(* CODESYS project Storage2018v1.project

Project tree, tasks and I/O mapping:
  CODESYS_Control_Win_V3_x64 : CODESYS Control Win V3 x64, 3S - Smart Software Solutions GmbH, version 3.5.12.30
    application Application
      libraries: BASIC, 3.31 (OSCAT)
      task VISU_TASK (cyclic, interval 50 ms, priority 31) calls VisuElems.Visu_Prg
      task Task (cyclic, interval t#20ms, priority 1) calls main, simulationLogic
      Control/
        program main [ST]
        Support/
          data type Position
          data type ArmRequest
          data type OPState
          function block ButtonRequester [LD]
          function PosToButtons [ST]
          function ButtonsToPos [ST]
          function block ArmRequestHandler [LD]
        program ArmControl [LD]
        function block PositionState [LD]
        function block OPArmMover [LD]
        function block OPGripper [SFC]
        function block OPPickNPlace [SFC]: copyVariables, gotoPos
        function block OPpnpTester [SFC]: setPick1, setPick2, setPick3, setPlace1, setPlace2, setPlace3
      doNotChange/
        Components/
          program simulationLogic [ST]
          visualisation armNStore
          Storage/
            visualisation StoragePlace
            visualisation Storage
            program storageLogic [ST]
          Conveyor/
            visualisation Conveyor
            program conveyorLogic [ST]
          Arm/
            visualisation TheArm
            program armLogic [ST]
            visualisation Gripper
        SimulationHelpers/
          function block MoveObject [ST]
        global variables InternalSimulation
        IO and DataTypes/
          data type CylPos
          data type XYPos
          data type ArmCommand
        internalTypes/
          data type StoragePos
        program simulationMapping [ST]
      Simulation/
        visualisation Simulation
      global variables IOs
  libraries: SysTimeCore, 3.5.5.0 (System)
  text list GlobalTextList
*)

// CODESYS_Control_Win_V3_x64/Application/Control/Support/Position
TYPE Position :
STRUCT
	x: INT;
	y: INT;
END_STRUCT
END_TYPE

// CODESYS_Control_Win_V3_x64/Application/Control/Support/ArmRequest
TYPE ArmRequest :
STRUCT
	run: BOOL;
	goto: Position;
END_STRUCT
END_TYPE

// CODESYS_Control_Win_V3_x64/Application/Control/Support/OPState
TYPE OPState :
STRUCT
	initial: BOOL;
	executing: BOOL;
	finished: BOOL;
END_STRUCT
END_TYPE

// CODESYS_Control_Win_V3_x64/Application/doNotChange/IO and DataTypes/CylPos
TYPE CylPos :
	STRUCT
		occupied: BOOL;
		id: STRING;
	END_STRUCT
END_TYPE

// CODESYS_Control_Win_V3_x64/Application/doNotChange/IO and DataTypes/XYPos
TYPE XYPos :
	STRUCT
		posX: INT;
		posY: INT;
	END_STRUCT
END_TYPE

// CODESYS_Control_Win_V3_x64/Application/doNotChange/IO and DataTypes/ArmCommand
TYPE ArmCommand :
STRUCT
	fromPos: XYPos;
	toPos: XYPos;
END_STRUCT
END_TYPE

// CODESYS_Control_Win_V3_x64/Application/doNotChange/internalTypes/StoragePos
TYPE StoragePos :
	STRUCT
		cyl: CylPos;
		pos: XYPos;
		pressed: Bool;
	END_STRUCT
END_TYPE

// CODESYS_Control_Win_V3_x64/Application/doNotChange/InternalSimulation
VAR_GLOBAL
	error: BOOL := FALSE;
	errorText: STRING := '';
	disablePressPos: BOOL := FALSE;
	buttonUP: BOOL;
	buttonDown: BOOL;
	buttonRun: BOOL;
	buttonDir: BOOL;
	buttonExt: BOOL;
	buttonRetr: BOOL;
	buttonGrip: BOOL;
END_VAR

// CODESYS_Control_Win_V3_x64/Application/IOs
VAR_GLOBAL
	qxArmRun: BOOL := FALSE; // Starts the arm moving left and right
	qxArmDirection: BOOL := FALSE; // true -> left, false -> right
	qxArmUp: BOOL := FALSE; // moves the arm up
	qxArmDown: BOOL := FALSE; // moves the arm down
	qxGripExtend: BOOL := FALSE; // extends the gripper
	qxGripRetract: BOOL := FALSE; // retracts the gripper
	qxGripping: BOOL := FALSE; // releases when false
	qxPosLamp: ARRAY[0..2, 0..2] OF BOOL;// lamp[X, Y] control if on / off
	
	ixArmAtX0: BOOL := FALSE;	// The arm postion
	ixArmAtX1: BOOL := FALSE;
	ixArmAtX2: BOOL := FALSE;
	ixArmAtY0: BOOL := FALSE;
	ixArmAtY1: BOOL := FALSE;
	ixArmAtY2: BOOL := FALSE;
	ixPosButtonDown: ARRAY[0..2, 0..2] OF BOOL;// Button[X, Y] is currently beeing pressed
	
	// These may not be the same as the qx versions above since the 
	// buttons in the simulation also can control the motion
	ixArmRun: BOOL := FALSE; // If the arm is moving left or rigth
	ixArmDirection: BOOL := FALSE; // true -> left, false -> right
	ixArmUp: BOOL := FALSE; // if arm is moving up
	ixArmDown: BOOL := FALSE; // if the arm is moving down
	
	ixGripExtended: BOOL := FALSE;	// the gripper has been extended
	ixGripRetracted: BOOL := FALSE; // the gripper has been retracted
	ixCylinderInGripper: BOOL:=FALSE; // A cylinder is carried by the arm
	
	ixEmergency: BOOL := TRUE; // Emergency stop if value is false
	ixStartButton: BOOL := FALSE;
	ixRunSequence: bool:= false;
		
END_VAR

// CODESYS_Control_Win_V3_x64/Application/Control/main
PROGRAM main
VAR

END_VAR

ArmControl();

END_PROGRAM

// CODESYS_Control_Win_V3_x64/Application/Control/ArmControl
PROGRAM ArmControl
VAR

	goto1: BOOL;
	goto0: BOOL;
	goto2: BOOL;
	
	initial: BOOL := FALSE;
	PositionStateY: PositionState;
	armYPosition: INT;
	armXPosition: INT;
	PositionStateX: PositionState;
	buttonReq: ButtonRequester;
	armMover: OPArmMover;
	moveRight: BOOL;
	moveLeft: BOOL;
	armGripper: OPGripper;
	reqHandler: ArmRequestHandler;
	pickNPlace: OPPickNPlace;
	staticPos: Position := (x := 3, y := 3);
	pnpTester: OPpnpTester;
END_VAR

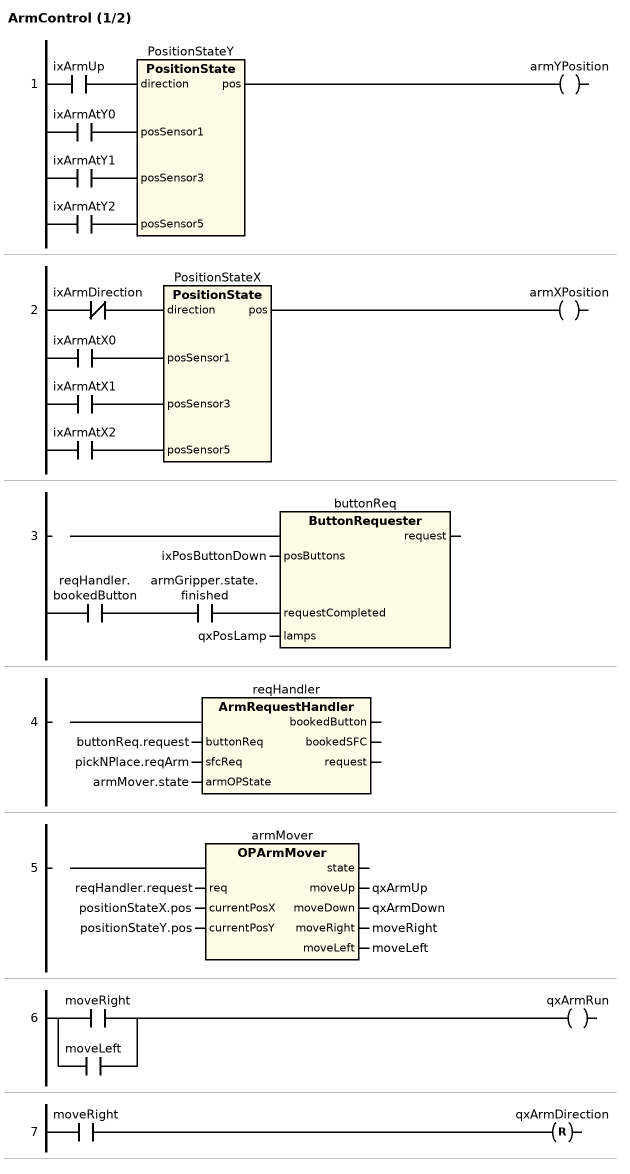
// NETWORK 1
PositionStateY(
    direction := ixArmUp,
    posSensor1 := ixArmAtY0,
    posSensor3 := ixArmAtY1,
    posSensor5 := ixArmAtY2); // PositionState
armYPosition := PositionStateY.pos;

// NETWORK 2
PositionStateX(
    direction := NOT ixArmDirection,
    posSensor1 := ixArmAtX0,
    posSensor3 := ixArmAtX1,
    posSensor5 := ixArmAtX2); // PositionState
armXPosition := PositionStateX.pos;

// NETWORK 3
buttonReq(
    posButtons := ixPosButtonDown,
    requestCompleted := reqHandler.bookedButton AND armGripper.state.finished,
    lamps := qxPosLamp); // ButtonRequester

// NETWORK 4
reqHandler(buttonReq := buttonReq.request, sfcReq := pickNPlace.reqArm, armOPState := armMover.state); // ArmRequestHandler

// NETWORK 5
armMover(
    req := reqHandler.request,
    currentPosX := positionStateX.pos,
    currentPosY := positionStateY.pos,
    moveUp => qxArmUp,
    moveDown => qxArmDown,
    moveRight => moveRight,
    moveLeft => moveLeft); // OPArmMover

// NETWORK 6
qxArmRun := moveRight OR moveLeft;

// NETWORK 7
qxArmDirection R= moveRight;

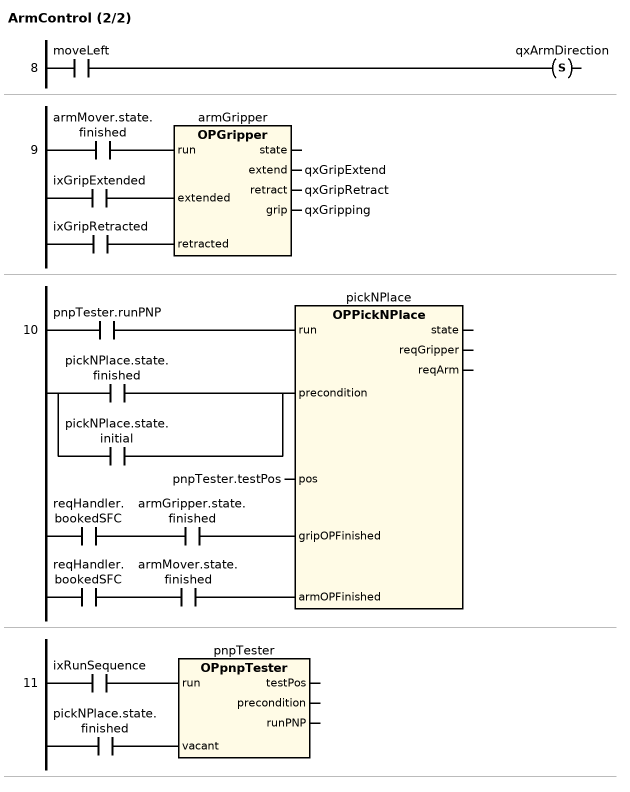
// NETWORK 8
qxArmDirection S= moveLeft;

// NETWORK 9
armGripper(
    run := armMover.state.finished,
    extended := ixGripExtended,
    retracted := ixGripRetracted,
    extend => qxGripExtend,
    retract => qxGripRetract,
    grip => qxGripping); // OPGripper

// NETWORK 10
pickNPlace(
    run := pnpTester.runPNP,
    precondition := pickNPlace.state.finished OR pickNPlace.state.initial,
    pos := pnpTester.testPos,
    gripOPFinished := reqHandler.bookedSFC AND armGripper.state.finished,
    armOPFinished := reqHandler.bookedSFC AND armMover.state.finished); // OPPickNPlace

// NETWORK 11
pnpTester(run := ixRunSequence, vacant := pickNPlace.state.finished); // OPpnpTester

END_PROGRAM

// CODESYS_Control_Win_V3_x64/Application/Control/PositionState
FUNCTION_BLOCK PositionState
VAR_INPUT
	direction: BOOL;
	posSensor1: BOOL;
	posSensor3: BOOL;
	posSensor5: BOOL;
END_VAR
VAR_OUTPUT
	pos: INT := -1;
END_VAR
VAR
	trig: F_TRIG;
END_VAR

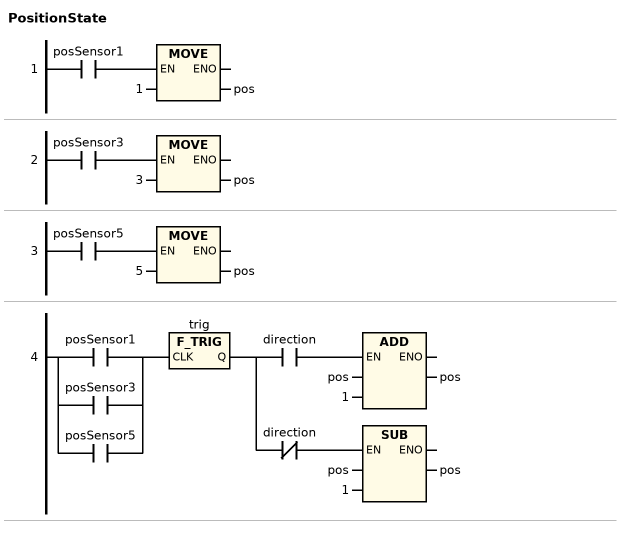
// NETWORK 1
IF posSensor1 THEN pos := 1; END_IF

// NETWORK 2
IF posSensor3 THEN pos := 3; END_IF

// NETWORK 3
IF posSensor5 THEN pos := 5; END_IF

// NETWORK 4
trig(CLK := posSensor1 OR posSensor3 OR posSensor5); // F_TRIG
IF trig.Q AND direction THEN pos := pos + 1; END_IF
IF trig.Q AND NOT direction THEN pos := pos - 1; END_IF

END_FUNCTION_BLOCK

// CODESYS_Control_Win_V3_x64/Application/Control/Support/ButtonRequester
FUNCTION_BLOCK ButtonRequester
VAR_INPUT
	posButtons: ARRAY[0..2, 0..2] OF BOOL;
	requestCompleted: BOOL;
END_VAR
VAR_OUTPUT
	request: ArmRequest;
END_VAR
VAR_IN_OUT
	lamps: ARRAY[0..2, 0..2] OF BOOL;
END_VAR

VAR
	armPos: Position;
	buttX: INT;
	buttY: INT;
	buttonPressed: BOOL;
	noRequest: ArmRequest := (run:=FALSE, goto := (x:=-1, y:=-1));
END_VAR
VAR // added by the converter: edge detectors and wires of the graphical bodies
    _w1 : BOOL;
END_VAR

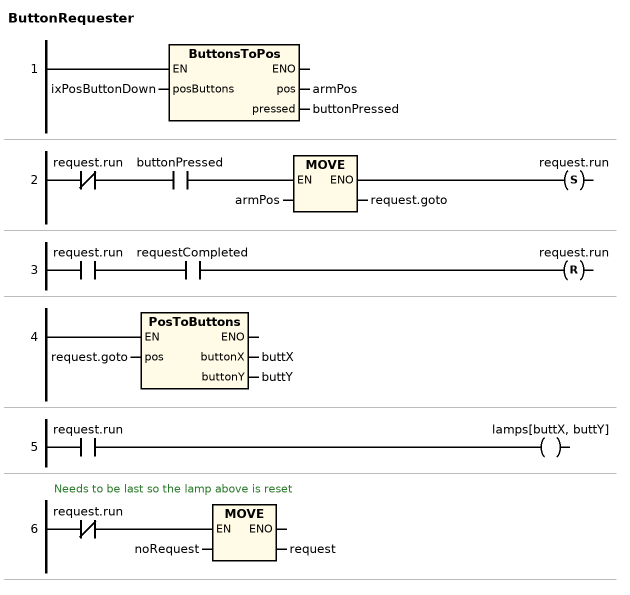
// NETWORK 1
ButtonsToPos(posButtons := ixPosButtonDown, pos => armPos, pressed => buttonPressed);

// NETWORK 2
_w1 := NOT request.run AND buttonPressed;
IF _w1 THEN request.goto := armPos; END_IF
request.run S= _w1;

// NETWORK 3
request.run R= request.run AND requestCompleted;

// NETWORK 4
PosToButtons(pos := request.goto, buttonX => buttX, buttonY => buttY);

// NETWORK 5
lamps[buttX, buttY] := request.run;

// NETWORK 6
// Needs to be last so the lamp above is reset
IF NOT request.run THEN request := noRequest; END_IF

END_FUNCTION_BLOCK

// CODESYS_Control_Win_V3_x64/Application/Control/Support/ButtonsToPos
FUNCTION ButtonsToPos
VAR_INPUT
	posButtons: ARRAY[0..2, 0..2] OF BOOL;
END_VAR
VAR_OUTPUT
	pos: Position;
	pressed: BOOL;
END_VAR
VAR
	x: INT;
	y: INT;
END_VAR

pos.x := -1;
pos.y := -1;
pressed := FALSE;

FOR x:=0 TO 2 DO
	FOR y:=0 TO 2 DO
		IF posButtons[x,y] THEN
			pos.x := 1 + x*2;
			pos.y := 1 + y*2;
			pressed := TRUE;
		END_IF
	END_FOR
END_FOR

END_FUNCTION

// CODESYS_Control_Win_V3_x64/Application/Control/Support/PosToButtons
FUNCTION PosToButtons
VAR_INPUT
	pos: Position;
END_VAR
VAR_OUTPUT
	buttonX: INT;
	buttonY: INT;
END_VAR
VAR
END_VAR

buttonX := -1;
buttonY := -1;
IF EVEN(pos.x-1) AND EVEN(pos.y-1) THEN
	buttonX:= (pos.x-1)/2;
	buttonY:= (pos.y-1)/2;
END_IF

END_FUNCTION

// CODESYS_Control_Win_V3_x64/Application/Control/Support/ArmRequestHandler
FUNCTION_BLOCK ArmRequestHandler
VAR_INPUT
	buttonReq: ArmRequest;
	sfcReq: ArmRequest;
	armOPState: OPState;
END_VAR
VAR_OUTPUT
	bookedButton: BOOL;
	bookedSFC: BOOL;
	request: ArmRequest;
END_VAR
VAR
	noRequest: ArmRequest := (run:=FALSE, goto := (x:=-1, y:=-1));
END_VAR

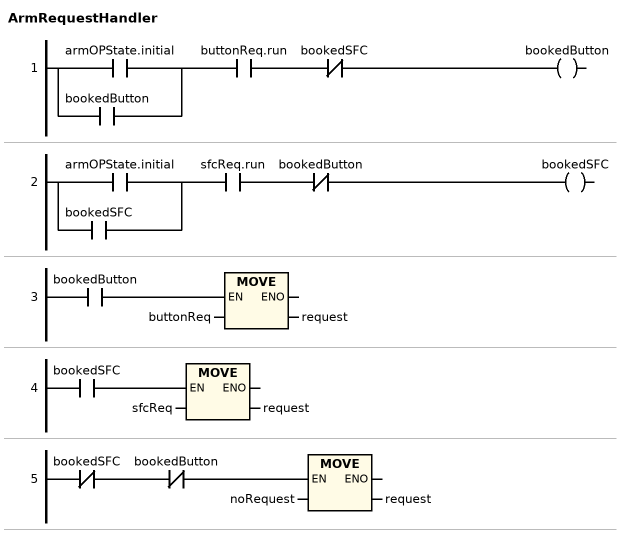
// NETWORK 1
bookedButton := (armOPState.initial OR bookedButton) AND buttonReq.run AND NOT bookedSFC;

// NETWORK 2
bookedSFC := (armOPState.initial OR bookedSFC) AND sfcReq.run AND NOT bookedButton;

// NETWORK 3
IF bookedButton THEN request := buttonReq; END_IF

// NETWORK 4
IF bookedSFC THEN request := sfcReq; END_IF

// NETWORK 5
IF NOT bookedSFC AND NOT bookedButton THEN request := noRequest; END_IF

END_FUNCTION_BLOCK

// CODESYS_Control_Win_V3_x64/Application/Control/OPArmMover
FUNCTION_BLOCK OPArmMover
VAR_INPUT
	req: ArmRequest;
	currentPosX: INT;
	currentPosY: INT;
END_VAR
VAR_OUTPUT
	state: OPState := (	initial := TRUE, 
						executing := FALSE, 
						finished := FALSE);
	moveUp: BOOL;
	moveDown: BOOL;
	moveRight: BOOL;
	moveLeft: BOOL;
END_VAR
VAR
	
	gotoX: INT;
	gotoY: INT;
	R_TRIG_0: R_TRIG;
	F_TRIG_0: F_TRIG;
	armGripper: OPGripper;
END_VAR
VAR // added by the converter: edge detectors and wires of the graphical bodies
    _w1, _w2 : BOOL;
END_VAR

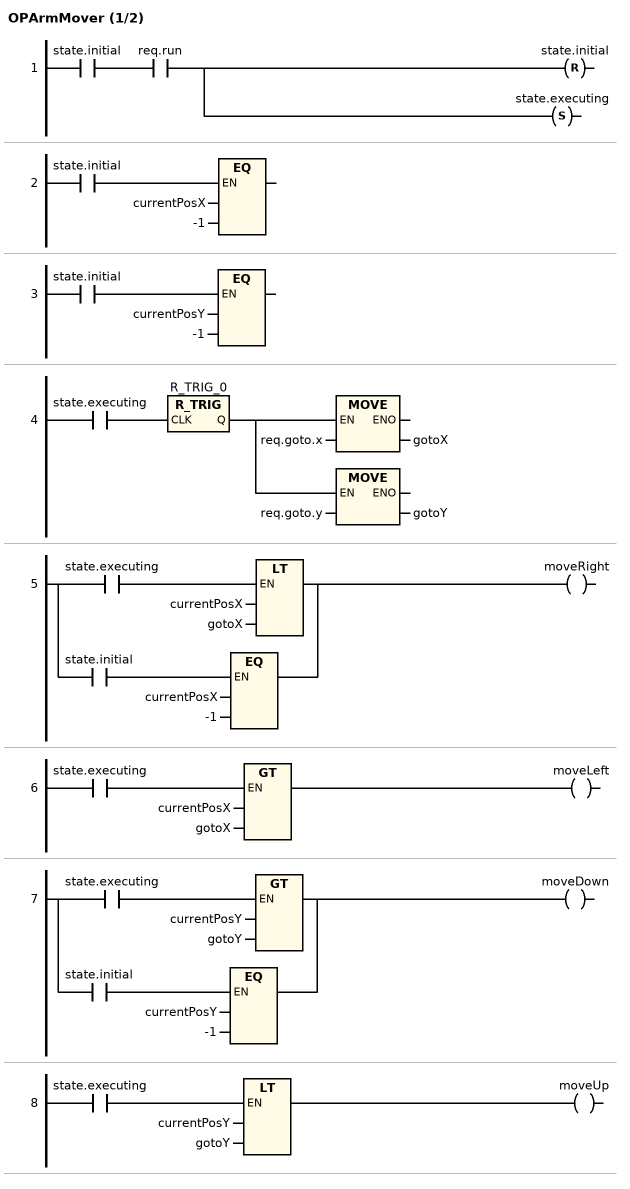
// NETWORK 1
_w1 := state.initial AND req.run;
state.initial R= _w1;
state.executing S= _w1;

// NETWORK 2
(* state.initial AND currentPosX = -1; result not used *)

// NETWORK 3
(* state.initial AND currentPosY = -1; result not used *)

// NETWORK 4
R_TRIG_0(CLK := state.executing); // R_TRIG
IF R_TRIG_0.Q THEN gotoX := req.goto.x; END_IF
IF R_TRIG_0.Q THEN gotoY := req.goto.y; END_IF

// NETWORK 5
moveRight := state.executing AND currentPosX < gotoX OR state.initial AND currentPosX = -1;

// NETWORK 6
moveLeft := state.executing AND currentPosX > gotoX;

// NETWORK 7
moveDown := state.executing AND currentPosY > gotoY OR state.initial AND currentPosY = -1;

// NETWORK 8
moveUp := state.executing AND currentPosY < gotoY;

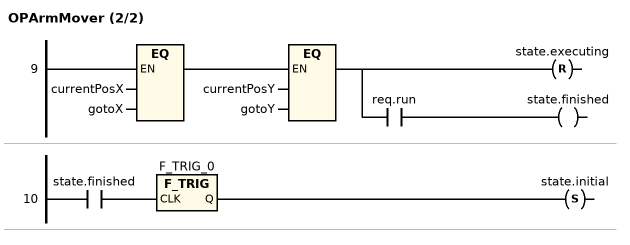
// NETWORK 9
_w2 := currentPosX = gotoX AND currentPosY = gotoY;
state.executing R= _w2;
state.finished := _w2 AND req.run;

// NETWORK 10
F_TRIG_0(CLK := state.finished); // F_TRIG
state.initial S= F_TRIG_0.Q;

END_FUNCTION_BLOCK

// CODESYS_Control_Win_V3_x64/Application/Control/OPGripper
FUNCTION_BLOCK OPGripper
VAR_INPUT
	run: BOOL;
	extended: BOOL;
	retracted: BOOL;
END_VAR
VAR_OUTPUT
	state: OPState;
	extend: BOOL;
	retract: BOOL;
	grip: BOOL;
END_VAR
VAR
END_VAR

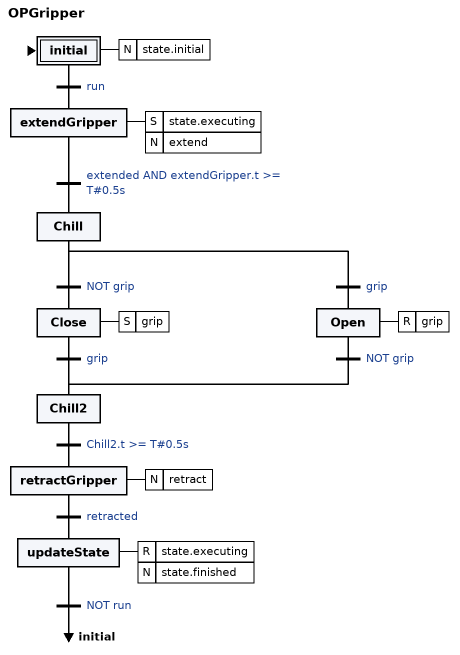
INITIAL_STEP initial:
    state.initial(N);
END_STEP
TRANSITION FROM initial TO extendGripper
    := run;
END_TRANSITION
STEP extendGripper:
    state.executing(S);
    extend(N);
END_STEP
TRANSITION FROM extendGripper TO Chill
    := extended AND extendGripper.t >= T#0.5s;
END_TRANSITION
STEP Chill:
END_STEP
TRANSITION FROM Chill TO Close
    := NOT grip;
END_TRANSITION
STEP Close:
    grip(S);
END_STEP
TRANSITION FROM Close TO Chill2
    := grip;
END_TRANSITION
TRANSITION FROM Chill TO Open
    := grip;
END_TRANSITION
STEP Open:
    grip(R);
END_STEP
TRANSITION FROM Open TO Chill2
    := NOT grip;
END_TRANSITION
STEP Chill2:
END_STEP
TRANSITION FROM Chill2 TO retractGripper
    := Chill2.t >= T#0.5s;
END_TRANSITION
STEP retractGripper:
    retract(N);
END_STEP
TRANSITION FROM retractGripper TO updateState
    := retracted;
END_TRANSITION
STEP updateState:
    state.executing(R);
    state.finished(N);
END_STEP
TRANSITION FROM updateState TO initial
    := NOT run;
END_TRANSITION

END_FUNCTION_BLOCK

// CODESYS_Control_Win_V3_x64/Application/Control/OPPickNPlace
FUNCTION_BLOCK OPPickNPlace
VAR_INPUT
	run: BOOL;
	precondition: BOOL;
	pos: Position;
	gripOPFinished: BOOL;
	armOPFinished: BOOL;
END_VAR
VAR_OUTPUT
	state: OPState;
	reqGripper: BOOL;
	reqArm: ArmRequest;
END_VAR
VAR
END_VAR

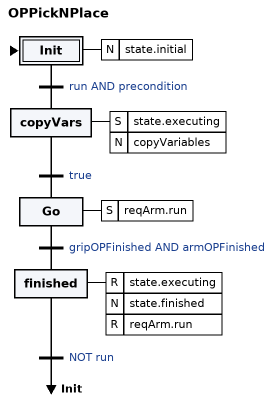
INITIAL_STEP Init:
    state.initial(N);
END_STEP
TRANSITION FROM Init TO copyVars
    := run AND precondition;
END_TRANSITION
STEP copyVars:
    state.executing(S);
    copyVariables(N);
END_STEP
TRANSITION FROM copyVars TO Go
    := true;
END_TRANSITION
STEP Go:
    reqArm.run(S);
END_STEP
TRANSITION FROM Go TO finished
    := gripOPFinished AND armOPFinished;
END_TRANSITION
STEP finished:
    state.executing(R);
    state.finished(N);
    reqArm.run(R);
END_STEP
TRANSITION FROM finished TO Init
    := NOT run;
END_TRANSITION

ACTION copyVariables:

(* Copy destination position *)
reqArm.goto.x := pos.x;
reqArm.goto.y := pos.y;
END_ACTION

ACTION gotoPos:
reqArm.run := true;
END_ACTION

END_FUNCTION_BLOCK

// CODESYS_Control_Win_V3_x64/Application/Control/OPpnpTester
FUNCTION_BLOCK OPpnpTester
VAR_INPUT
	run: BOOL;
	vacant: BOOL;
END_VAR
VAR_OUTPUT
	testPos: Position;
	precondition: BOOL;
	runPNP: BOOL;
END_VAR
VAR
	pick1: Position := (x := 1, y := 3);
	place1: Position := (x := 5, y := 5);
	
	pick2: Position := (x := 5, y := 1);
	place2: Position := (x := 3, y := 3);
	
	pick3: Position := (x := 3, y := 3);
	place3: Position := (x := 1, y := 5);
END_VAR

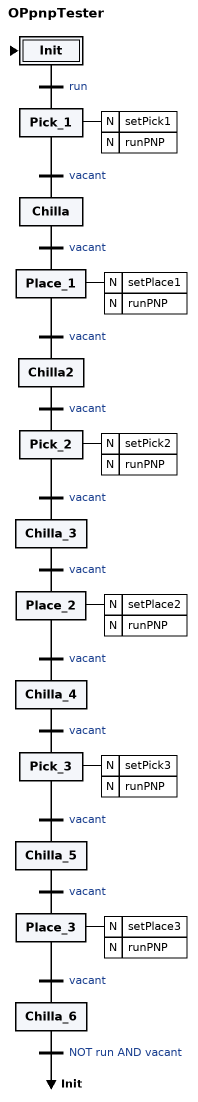
INITIAL_STEP Init:
END_STEP
TRANSITION FROM Init TO Pick_1
    := run;
END_TRANSITION
STEP Pick_1:
    setPick1(N);
    runPNP(N);
END_STEP
TRANSITION FROM Pick_1 TO Chilla
    := vacant;
END_TRANSITION
STEP Chilla:
END_STEP
TRANSITION FROM Chilla TO Place_1
    := vacant;
END_TRANSITION
STEP Place_1:
    setPlace1(N);
    runPNP(N);
END_STEP
TRANSITION FROM Place_1 TO Chilla2
    := vacant;
END_TRANSITION
STEP Chilla2:
END_STEP
TRANSITION FROM Chilla2 TO Pick_2
    := vacant;
END_TRANSITION
STEP Pick_2:
    setPick2(N);
    runPNP(N);
END_STEP
TRANSITION FROM Pick_2 TO Chilla_3
    := vacant;
END_TRANSITION
STEP Chilla_3:
END_STEP
TRANSITION FROM Chilla_3 TO Place_2
    := vacant;
END_TRANSITION
STEP Place_2:
    setPlace2(N);
    runPNP(N);
END_STEP
TRANSITION FROM Place_2 TO Chilla_4
    := vacant;
END_TRANSITION
STEP Chilla_4:
END_STEP
TRANSITION FROM Chilla_4 TO Pick_3
    := vacant;
END_TRANSITION
STEP Pick_3:
    setPick3(N);
    runPNP(N);
END_STEP
TRANSITION FROM Pick_3 TO Chilla_5
    := vacant;
END_TRANSITION
STEP Chilla_5:
END_STEP
TRANSITION FROM Chilla_5 TO Place_3
    := vacant;
END_TRANSITION
STEP Place_3:
    setPlace3(N);
    runPNP(N);
END_STEP
TRANSITION FROM Place_3 TO Chilla_6
    := vacant;
END_TRANSITION
STEP Chilla_6:
END_STEP
TRANSITION FROM Chilla_6 TO Init
    := NOT run AND vacant;
END_TRANSITION

ACTION setPick1:


testPos.x := pick1.x;
testPos.y := pick1.y;
END_ACTION

ACTION setPick2:


testPos.x := pick2.x;
testPos.y := pick2.y;
END_ACTION

ACTION setPick3:


testPos.x := pick3.x;
testPos.y := pick3.y;
END_ACTION

ACTION setPlace1:


testPos.x := place1.x;
testPos.y := place1.y;
END_ACTION

ACTION setPlace2:


testPos.x := place2.x;
testPos.y := place2.y;
END_ACTION

ACTION setPlace3:


testPos.x := place3.x;
testPos.y := place3.y;
END_ACTION

END_FUNCTION_BLOCK

// CODESYS_Control_Win_V3_x64/Application/doNotChange/Components/simulationLogic
PROGRAM simulationLogic
VAR
	armAtX0: BOOL := FALSE;
	armAtX1: BOOL := FALSE;
	armAtX2: BOOL := FALSE;
	armAtY0: BOOL := FALSE;
	armAtY1: BOOL := FALSE;
	armAtY2: BOOL := FALSE;
	inAnyPos: BOOL := FALSE;
	graspTrig: R_TRIG;
	relTrig: F_TRIG;
	grasp: BOOL;
	release: BOOL;
	errorMsg: STRING := '';
	ack: BOOL:= FALSE;
	e_stop: BOOL:= FALSE;
	allowPick: BOOL;
END_VAR

storageLogic();
armLogic();
simulationMapping();

armAtX0 := armLogic.armPosX > 90 AND armLogic.armPosX < 95;
armAtX1 := armLogic.armPosX > 205 AND armLogic.armPosX < 210;
armAtX2 := armLogic.armPosX > 320 AND armLogic.armPosX < 325;

armAtY2 := armLogic.armPosY > 0 AND armLogic.armPosY < 15;
armAtY1 := armLogic.armPosY > 100 AND armLogic.armPosY < 115;
armAtY0 := armLogic.armPosY > 200 AND armLogic.armPosY < 215;

inAnyPos := (armAtX0 OR armAtX1 OR armAtX2) AND (armAtY0 OR armAtY1 OR armAtY2);
allowPick := inAnyPos AND ixGripExtended;

graspTrig(CLK:= qxGripping, Q=> grasp);
relTrig(CLK:= qxGripping, Q=> release);

IF grasp AND allowPick THEN
	ixCylinderInGripper := TRUE;
END_IF
IF release AND allowPick THEN
	ixCylinderInGripper := FALSE;
END_IF

// Error handling
IF e_stop AND ixEmergency THEN
	ixEmergency := FALSE;
	errorMsg := 'You pressed the Emergency';
END_IF
IF ack THEN
	ixEmergency := TRUE;
	errorMsg := '';
END_IF

IF grasp AND inAnyPos AND NOT allowPick AND ixEmergency THEN
	ixEmergency := FALSE;
	errorMsg := 'Not grasping when gripper is extended!';
ELSIF grasp AND NOT inAnyPos AND ixEmergency THEN
	ixEmergency := FALSE;
	errorMsg := 'Not grasping at a XY position!';
END_IF

IF release AND (NOT inAnyPos OR NOT ixGripExtended) AND ixEmergency AND ixCylinderInGripper THEN
	ixEmergency := FALSE;
	errorMsg := 'You dropped the cylinder';
	ixCylinderInGripper := FALSE;
END_IF

IF (qxArmRun OR qxArmDown OR qxArmUp) AND ixGripExtended THEN
	ixEmergency := FALSE;
	errorMsg := 'Can not move white extended gripper';
END_IF

END_PROGRAM

// CODESYS_Control_Win_V3_x64/Application/doNotChange/Components/Storage/storageLogic
PROGRAM storageLogic
VAR
	storagePlaces: ARRAY[0..2, 0..2] OF StoragePos;
END_VAR

	storageLogic.storagePlaces[0,0].cyl.occupied := qxPosLamp[0,0];
	storageLogic.storagePlaces[0,1].cyl.occupied := qxPosLamp[0,1];
	storageLogic.storagePlaces[0,2].cyl.occupied := qxPosLamp[0,2];
	storageLogic.storagePlaces[1,0].cyl.occupied := qxPosLamp[1,0];
	storageLogic.storagePlaces[1,1].cyl.occupied := qxPosLamp[1,1];
	storageLogic.storagePlaces[1,2].cyl.occupied := qxPosLamp[1,2];
	storageLogic.storagePlaces[2,0].cyl.occupied := qxPosLamp[2,0];
	storageLogic.storagePlaces[2,1].cyl.occupied := qxPosLamp[2,1];
	storageLogic.storagePlaces[2,2].cyl.occupied := qxPosLamp[2,2];

END_PROGRAM

// CODESYS_Control_Win_V3_x64/Application/doNotChange/Components/Arm/armLogic
PROGRAM armLogic
VAR
	gripping: BOOL := FALSE;
	extending: BOOL := FALSE;
	cyl: CylPos := (occupied := FALSE, id:= '');
	armPosX : INT;
	armPosY : INT;
	gripYPos: INT := 0;
	gripXPos: INT := 0;
	moveArm: MoveObject;
	armDown: BOOL := FALSE;
	armUP: BOOL := false;
	armL: BOOL := false;
	armR: BOOL := false;
END_VAR
VAR_TEMP
	
END_VAR

IF extending THEN
	gripYPos := -25;
ELSE
	gripYPos := 0;
END_IF
gripXPos := 0;

armLogic.cyl.occupied := ixCylinderInGripper;
IF ixCylinderInGripper THEN
	armLogic.cyl.id := 'Cylinder';
ELSE
	armLogic.cyl.id := '';
END_IF

moveArm(
	moveUP:= armUP, 
	moveDown:= armDown, 
	moveLeft:=armL , 
	moveRight:=armR , 
	maxX:=400, 
	minX:=0, 
	maxY:=220, 
	minY:=0, 
	tick:=T#0.01S , 
	x:= armPosX, 
	y:=armPosY );
	
	armLogic.armR := (qxArmRun AND NOT qxArmDirection) OR (buttonRun AND NOT buttonDir) ;
	armLogic.armL := (qxArmRun AND qxArmDirection) OR (buttonRun AND buttonDir);	
	armLogic.armUP := qxArmUp OR buttonUP;
	armLogic.armDown := qxArmDown OR buttonDown;
	armLogic.extending := qxGripExtend OR buttonExt OR (armLogic.extending AND NOT (qxGripRetract OR buttonRetr));
	armLogic.gripping := qxGripping OR buttonGrip;
	
	ixArmUp := armLogic.armUP;
	ixArmDown := armLogic.armDown;
	ixArmRun := qxArmRun OR buttonRun;
	ixArmDirection := qxArmDirection OR buttonDir;

END_PROGRAM

// CODESYS_Control_Win_V3_x64/Application/doNotChange/SimulationHelpers/MoveObject
FUNCTION_BLOCK MoveObject
VAR_INPUT
	moveUP: BOOL;
	moveDown: BOOL;
	moveLeft: BOOL;
	moveRight: BOOL;
	maxX: INT;
	minX: INT;
	maxY: INT;
	minY: INT;
	tick: time;
END_VAR
VAR_IN_OUT
	x: INT;
	y: INT;
END_VAR
VAR_OUTPUT
END_VAR
VAR
	pulse: clk_pulse;
END_VAR

pulse(
	PT:= tick, 
	N:= 0, 
	RST:= NOT moveUp AND NOT moveDown AND NOT moveLeft AND NOT moveRight , 
	Q=> , 
	CNT=> , 
	RUN=> );
	
IF pulse.Q THEN
	IF moveUP AND NOT moveDown AND y > minY THEN
		y := y-1;
	ELSIF NOT moveUP AND moveDown AND y < maxY THEN
		y := y+1;
	END_IF
	
	IF moveRight AND NOT moveLeft AND x < maxX THEN
		x := x+1;
	ELSIF NOT moveRight AND moveLeft AND x > minX THEN
		x := x-1;
	END_IF
END_IF

END_FUNCTION_BLOCK

// CODESYS_Control_Win_V3_x64/Application/doNotChange/simulationMapping
PROGRAM simulationMapping
VAR
END_VAR



	

	
	
	ixArmAtX0 := simulationLogic.armAtX0;
	ixArmAtX1 := simulationLogic.armAtX1;
	ixArmAtX2 := simulationLogic.armAtX2;
	ixArmAtY0 := simulationLogic.armAtY0;
	ixArmAtY1 := simulationLogic.armAtY1;
	ixArmAtY2 := simulationLogic.armAtY2;
	ixPosButtonDown[0,0] := storageLogic.storagePlaces[0,0].pressed;
	ixPosButtonDown[0,1] := storageLogic.storagePlaces[0,1].pressed;
	ixPosButtonDown[0,2] := storageLogic.storagePlaces[0,2].pressed;
	ixPosButtonDown[1,0] := storageLogic.storagePlaces[1,0].pressed;
	ixPosButtonDown[1,1] := storageLogic.storagePlaces[1,1].pressed;
	ixPosButtonDown[1,2] := storageLogic.storagePlaces[1,2].pressed;
	ixPosButtonDown[2,0] := storageLogic.storagePlaces[2,0].pressed;
	ixPosButtonDown[2,1] := storageLogic.storagePlaces[2,1].pressed;
	ixPosButtonDown[2,2] := storageLogic.storagePlaces[2,2].pressed;
	
	ixGripExtended := armLogic.extending;
	ixGripRetracted := NOT armLogic.extending;
	
	
	
	// use as is ixEmergency
	// use as is ixStartButton

END_PROGRAM

// CODESYS_Control_Win_V3_x64/Application/doNotChange/Components/Conveyor/conveyorLogic
PROGRAM conveyorLogic
VAR
	places: ARRAY[0..7] OF StoragePos;
	inSensor: BOOL := FALSE;
	outSensor: BOOL := FALSE;
	run: BOOL := FALSE;
	dir: BOOL := FALSE; 
END_VAR

END_PROGRAM

// CODESYS_Control_Win_V3_x64/Application/doNotChange/Components/armNStore
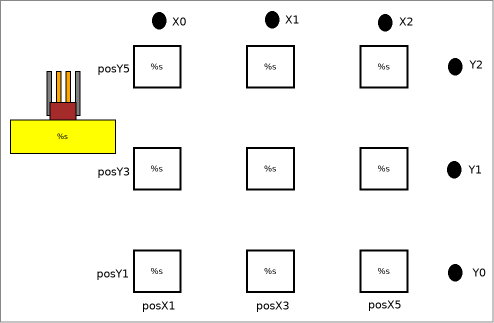
VISUALIZATION armNStore  // 494x323
    Frame (133,45 277x250)
        shows Storage()
    Ellipse (448,58 14x17), colour toggle: simulationLogic.armAtY2
    Ellipse (447,161 14x17), colour toggle: simulationLogic.armAtY1
    Ellipse (448,264 14x17), colour toggle: simulationLogic.armAtY0
    Ellipse (152,12 14x17), colour toggle: simulationLogic.armAtX0
    Ellipse (265,11 14x17), colour toggle: simulationLogic.armAtX1
    Ellipse (378,14 14x17), colour toggle: simulationLogic.armAtX2
    Label (167,7 25x30), "X0"
    Label (280,5 25x30), "X1"
    Label (394,7 25x30), "X2"
    Label (467,258 25x30), "Y0"
    Label (463,155 25x30), "Y1"
    Label (464,50 25x30), "Y2"
    Frame (10,54 107x101)
        shows TheArm()
        p3560616238: armLogic.armPosX
        p2738717112: armLogic.armPosY
    Label (138,291 42x30), "posX1"
    Label (252,291 42x30), "posX3"
    Label (364,290 42x30), "posX5"
    Label (83,261 60x26), "posY1"
    Label (84,159 60x26), "posY3"
    Label (84,56 60x26), "posY5"
END_VISUALIZATION

// CODESYS_Control_Win_V3_x64/Application/doNotChange/Components/Storage/StoragePlace
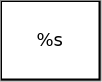
VISUALIZATION StoragePlace  // 102x82
VAR_IN_OUT
	pos: StoragePos;
END_VAR
    Rectangle (0,0 100x80), "%s", text variable: pos.cyl.id, colour toggle: pos.cyl.occupied
        tap pos.pressed
END_VISUALIZATION

// CODESYS_Control_Win_V3_x64/Application/doNotChange/Components/Storage/Storage
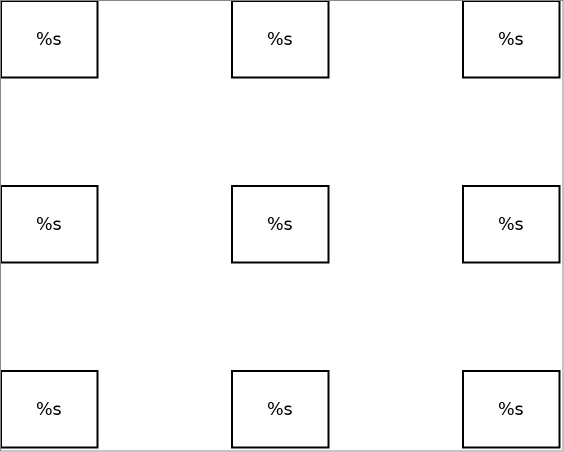
VISUALIZATION Storage  // 564x452
    Frame (0,370 100x80)
        shows StoragePlace(pos := storageLogic.storagePlaces[0, 0])
    Frame (0,185 100x80)
        shows StoragePlace(pos := storageLogic.storagePlaces[0, 1])
    Frame (0,0 100x80)
        shows StoragePlace(pos := storageLogic.storagePlaces[0, 2])
    Frame (231,370 100x80)
        shows StoragePlace(pos := storageLogic.storagePlaces[1, 0])
    Frame (231,185 100x80)
        shows StoragePlace(pos := storageLogic.storagePlaces[1, 1])
    Frame (231,0 100x80)
        shows StoragePlace(pos := storageLogic.storagePlaces[1,2])
    Frame (462,370 100x80)
        shows StoragePlace(pos := storageLogic.storagePlaces[2, 0])
    Frame (462,185 100x80)
        shows StoragePlace(pos := storageLogic.storagePlaces[2, 1])
    Frame (462,0 100x80)
        shows StoragePlace(pos := storageLogic.storagePlaces[2,2])
END_VISUALIZATION

// CODESYS_Control_Win_V3_x64/Application/doNotChange/Components/Conveyor/Conveyor
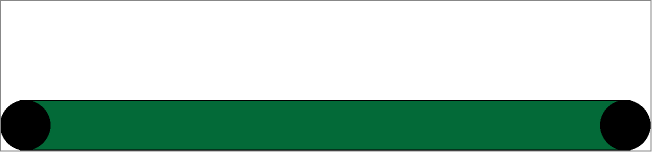
VISUALIZATION Conveyor  // 652x152
    RoundedRectangle (20,100 610x50)
    Ellipse (0,100 50x50), colour toggle: conveyorLogic.run and conveyorLogic.dir
    Ellipse (600,100 50x50), colour toggle: conveyorLogic.run and not conveyorLogic.dir
END_VISUALIZATION

// CODESYS_Control_Win_V3_x64/Application/doNotChange/Components/Arm/TheArm
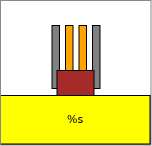
VISUALIZATION TheArm  // 152x146
    Frame (48,25 54x109)
        shows Gripper(gripping := armLogic.gripping)
        p2738717112: armLogic.gripYPos
        p3560616238: armLogic.gripXPos
    RoundedRectangle (0,95 150x49), "%s", text variable: armLogic.cyl.id, colour toggle: armLogic.cyl.occupied
END_VISUALIZATION

// CODESYS_Control_Win_V3_x64/Application/doNotChange/Components/Arm/Gripper
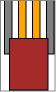
VISUALIZATION Gripper  // 56x92
VAR_IN_OUT
	gripping: bool;
END_VAR
    Group (4,0 50x40), invisible if: gripping
        Rectangle (0,0 8x54)
        Rectangle (42,0 8x54)
    Group (18,0 22x39), invisible if: not gripping
        Rectangle (0,0 8x54)
        Rectangle (14,0 8x54)
    Rectangle (9,38 39x52)
END_VISUALIZATION

// CODESYS_Control_Win_V3_x64/Application/Simulation/Simulation
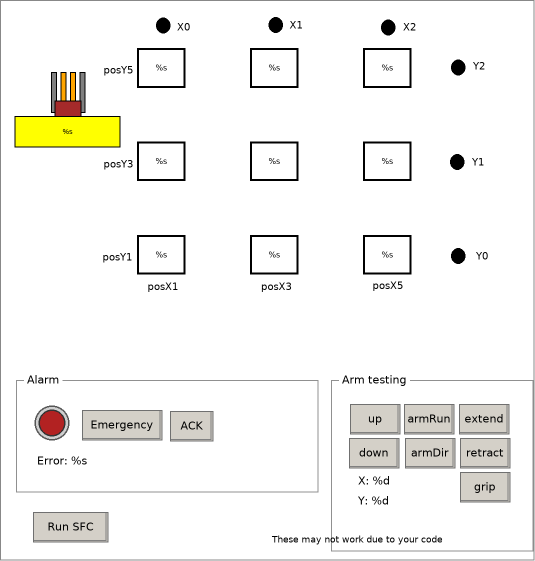
VISUALIZATION Simulation  // 535x561
    GroupBox (331,372 202x179), "Arm testing"
        Button (19,32 50x30), "up"
            toggle buttonUP
        Button (18,66 50x30), "down"
            toggle buttonDown
        Button (73,32 50x30), "armRun"
            toggle buttonRun
        Button (74,66 50x30), "armDir"
            toggle buttonDir
        Button (128,32 50x30), "extend"
            toggle buttonExt
        Button (129,66 50x30), "retract"
            toggle buttonRetr
        Button (129,100 50x30), "grip"
            toggle buttonGrip
    Rectangle (355,469 100x24), "X: %d", text variable: armLogic.armPosX
    Rectangle (355,489 100x24), "Y: %d", text variable: armLogic.armPosY
    Frame (5,7 492x295)
        shows armNStore()
    GroupBox (16,372 302x120), "Alarm"
        Lamp1 (15,31 42x40), variable: not ixEmergency, style: Lamp-Lamp1-Red
        Rectangle (18,72 268x34), "Error: %s", text variable: simulationLogic.errorMsg, invisible if: ixEmergency
        Button (66,38 80x30), "Emergency"
            tap simulationLogic.e_stop
        Button (154,39 43x30), "ACK"
            tap simulationLogic.ack
        Button (17,140 75x30), "Run SFC"
            tap ixRunSequence
    Label (256,520 203x39), "These may not work due to your code"
END_VISUALIZATION
